PROGRAM MAIN
VAR

	M1 : DUT_MotionStage := (nEnableMode:=ENUM_StageEnableMode.ALWAYS, bPowerSelf:=TRUE);
    fbMotionStageM1 : FB_MotionStage;
END_VAR

fbMotionStageM1(stMotionStage:=M1);
m1.bHardwareEnable := True;
m1.bLimitBackwardEnable := True;
m1.bLimitForwardEnable := True;

END_PROGRAM

(* stored: Version 1.1.0.1, ProductVersion 3.1.4022.18
   POU MAIN: Id {78820bd1-5267-489e-8f09-6a788ae2c68a}, SpecialFunc None *)
